// TIA Portal V18 export
FUNCTION_BLOCK "Initial_Test_Squence"   // FB18, LAD
{ S7_Optimized_Access := 'TRUE' }
VERSION : 0.1
// stored: AutoNumber true, IsIECCheckEnabled false, IsRetainMemResEnabled false, MemoryReserve 100, SetENOAutomatically false, UDAEnableTagReadback false
   VAR_INPUT
      ON : Bool;
      Position : DInt;
      HomingOK : Bool;
      InputTask : Bool;
      StepSizeInput : DInt := 100;
      AmountOfSteps : Int := 100;
   END_VAR
   VAR_OUTPUT
      StartMachine : Bool;
      StartHoming : Bool;
      StepSizeOutput : DInt := 1000;
      TestFinished : Bool;
      StartPosition : DInt;
      EndPositon : DInt;
   END_VAR
   VAR_IN_OUT
      StartTask : Bool;
   END_VAR
   VAR
      TurnOnM : Bool;
      StepNumber : Int;
      InternalWait { ExternalAccessible := 'False'; ExternalVisible := 'False'; ExternalWritable := 'False'} : Bool;
      StepNumberNext { ExternalAccessible := 'False'; ExternalVisible := 'False'; ExternalWritable := 'False'} : Int;
      ONM : Bool;
      TestFinishedM : Bool;
      StartTaskM { ExternalAccessible := 'False'; ExternalVisible := 'False'; ExternalWritable := 'False'} : Bool;
   END_VAR
   VAR_TEMP   // added for the SCL form of the ladder/FBD networks
      _w1 : Bool;
   END_VAR
BEGIN

REGION Network 1: Turn On
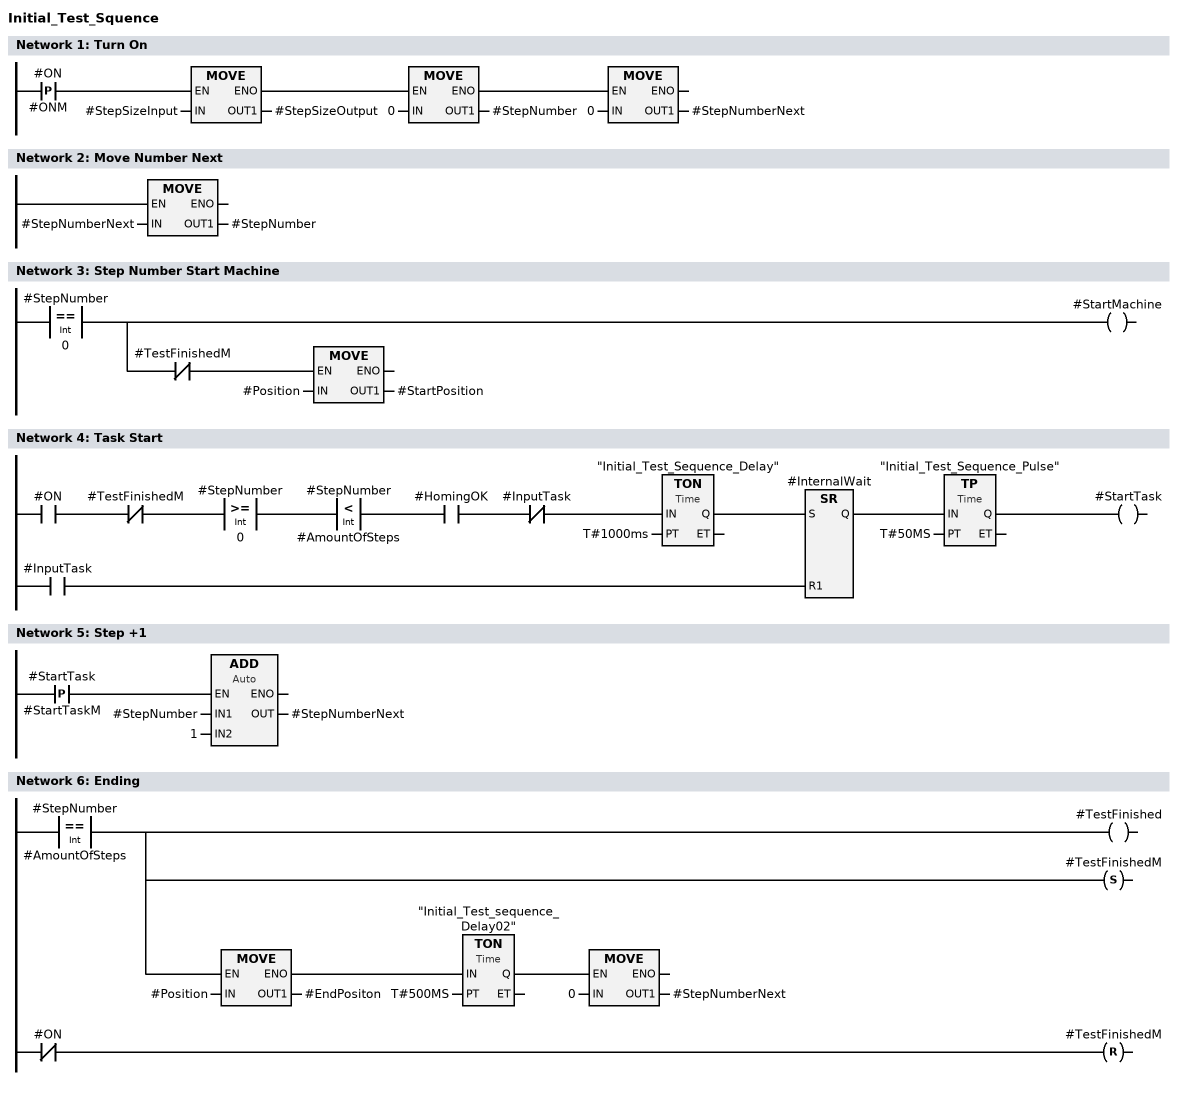
   RUNG wire#powerrail
      P_Contact(operand := #ON, bit := #ONM)
      Move(in := #StepSizeInput, out1 => #StepSizeOutput)
      Move(in := 0, out1 => #StepNumber)
      Move(in := 0, out1 => #StepNumberNext)
   END_RUNG
   // the same network as SCL:
   #_w1 := #ON AND NOT #ONM;   // rising edge of #ON
   #ONM := #ON;
   IF #_w1 THEN
       #StepSizeOutput := #StepSizeInput;
       #StepNumber := 0;
       #StepNumberNext := 0;
   END_IF;
END_REGION

REGION Network 2: Move Number Next
   RUNG wire#powerrail
      Move(in := #StepNumberNext, out1 => #StepNumber)
   END_RUNG
   // the same network as SCL:
   #StepNumber := #StepNumberNext;
END_REGION

REGION Network 3: Step Number Start Machine
   RUNG wire#powerrail
      { S7_Templates := "SrcType := Int" } EQ_Contact(in1 := #StepNumber, in2 := 0)
      wire#w1
      Coil( #StartMachine )
   END_RUNG
   RUNG wire#w1
      I_Contact( #TestFinishedM )
      Move(in := #Position, out1 => #StartPosition)
   END_RUNG
   // the same network as SCL:
   #StartMachine := #StepNumber = 0;
   IF #StartMachine AND NOT #TestFinishedM THEN #StartPosition := #Position; END_IF;
END_REGION

REGION Network 4: Task Start
   RUNG wire#powerrail
      Contact( #ON )
      I_Contact( #TestFinishedM )
      { S7_Templates := "SrcType := Int" } GE_Contact(in1 := #StepNumber, in2 := 0)
      { S7_Templates := "SrcType := Int" } LT_Contact(in1 := #StepNumber, in2 := #AmountOfSteps)
      Contact( #HomingOK )
      I_Contact( #InputTask )
      { S7_Templates := "time_type := Time" } "Initial_Test_Sequence_Delay".TON(pt := T#1000ms, et =>)
      S_SR(operand := #InternalWait, r1 := wire#w1)
      { S7_Templates := "time_type := Time" } "Initial_Test_Sequence_Pulse".TP(pt := T#50MS, et =>)
      Coil( #StartTask )
   END_RUNG
   RUNG wire#powerrail
      Contact( #InputTask )
   END_RUNG wire#w1
   // the same network as SCL:
   "Initial_Test_Sequence_Delay".TON(IN := #ON AND NOT #TestFinishedM AND (#StepNumber >= 0) AND (#StepNumber < #AmountOfSteps) AND #HomingOK AND NOT #InputTask,
                           PT := T#1000ms);
   IF "Initial_Test_Sequence_Delay".Q THEN
       #InternalWait := TRUE;   // SR flip-flop
   END_IF;
   IF #InputTask THEN #InternalWait := FALSE; END_IF;
   "Initial_Test_Sequence_Pulse".TP(IN := #InternalWait, PT := T#50MS);
   #StartTask := "Initial_Test_Sequence_Pulse".Q;
END_REGION

REGION Network 5: Step +1
   RUNG wire#powerrail
      P_Contact(operand := #StartTask, bit := #StartTaskM)
      Add(in1 := #StepNumber, in2 := 1, out => #StepNumberNext)
   END_RUNG
   // the same network as SCL:
   #_w1 := #StartTask AND NOT #StartTaskM;   // rising edge of #StartTask
   #StartTaskM := #StartTask;
   IF #_w1 THEN #StepNumberNext := #StepNumber + 1; END_IF;
END_REGION

REGION Network 6: Ending
   RUNG wire#powerrail
      { S7_Templates := "SrcType := Int" } EQ_Contact(in1 := #StepNumber, in2 := #AmountOfSteps)
      wire#w1
      Coil( #TestFinished )
   END_RUNG
   RUNG wire#w1
      S_Coil( #TestFinishedM )
   END_RUNG
   RUNG wire#w1
      Move(in := #Position, out1 => #EndPositon)
      { S7_Templates := "time_type := Time" } "Initial_Test_sequence_Delay02".TON(pt := T#500MS, et =>)
      Move(in := 0, out1 => #StepNumberNext)
   END_RUNG
   RUNG wire#powerrail
      I_Contact( #ON )
      R_Coil( #TestFinishedM )
   END_RUNG
   // the same network as SCL:
   #TestFinished := #StepNumber = #AmountOfSteps;
   IF #TestFinished THEN
       #TestFinishedM := TRUE;
       #EndPositon := #Position;
   END_IF;
   "Initial_Test_sequence_Delay02".TON(IN := #TestFinished, PT := T#500MS);
   IF "Initial_Test_sequence_Delay02".Q THEN #StepNumberNext := 0; END_IF;
   IF NOT #ON THEN #TestFinishedM := FALSE; END_IF;
END_REGION
END_FUNCTION_BLOCK
